// TIA Portal V15.1 export
// export: Created 2024-06-21T08:40:52.8738255Z, ExportSetting WithDefaults, DisplayName Totally Integrated Automation Portal, DisplayVersion V15.1 Update 5, DisplayName TIA Portal Openness, DisplayVersion V15.1 Update 5, DisplayName SINAMICS Startdrive Advanced, DisplayVersion V15.1, DisplayName G130, G150, S120, S150, SINAMICS MV, S210, DisplayVersion V15.1, DisplayName G110M, G120, G120C, G120D, G120P, DisplayVersion V15.1, DisplayName STEP 7 Professional, DisplayVersion V15.1 Update 5, DisplayName STEP 7 Safety, DisplayVersion V15.1, DisplayName WinCC Professional, DisplayVersion V15.1 Update 5, DisplayName SIMATIC Visualization Architect, DisplayVersion V15.1
FUNCTION_BLOCK "LGeneralReverse"   // FB1103, FBD
TITLE = LGeneralReverse
{ S7_Optimized_Access := 'TRUE' }
VERSION : 0.1
// stored: AutoNumber false, IsIECCheckEnabled false, IsRetainMemResEnabled false, MemoryReserve 100, SetENOAutomatically False, UDAEnableTagReadback false
   VAR_INPUT
      I_GeneralReverseSw { ExternalAccessible := 'False'; ExternalVisible := 'False'; ExternalWritable := 'False'} : Bool;   // General reverse switch
      I_FbkContactorFwd { ExternalAccessible := 'False'; ExternalVisible := 'False'; ExternalWritable := 'False'} : Bool;   // Feedback contactor Forward
      I_FbkContactorBwd { ExternalAccessible := 'False'; ExternalVisible := 'False'; ExternalWritable := 'False'} : Bool;   // Feedback contactor Backward
      I_EnableAlarm { ExternalAccessible := 'False'; ExternalVisible := 'False'; ExternalWritable := 'False'} : Bool;   // Enable alarm / Enable Alarm
      I_ResetFbkAlarm { ExternalAccessible := 'False'; ExternalVisible := 'False'; ExternalWritable := 'False'} : Bool;   // Reset feedback alarm / Alarm reset pushbutton is activated
      C_FeedbackUsed { ExternalAccessible := 'False'; ExternalVisible := 'False'; ExternalWritable := 'False'} : Bool;   // Config Feedback used
   END_VAR
   VAR_OUTPUT
      O_ContactorFwd { ExternalAccessible := 'False'; ExternalVisible := 'False'; ExternalWritable := 'False'} : Bool;   // Activate low speed contactor / Activate Forward contactor
      O_ContactorBwd { ExternalAccessible := 'False'; ExternalVisible := 'False'; ExternalWritable := 'False'} : Bool;   // Activate High Speed contactor / Activate Backward contactor
      O_GenRevSw { ExternalAccessible := 'False'; ExternalVisible := 'False'; ExternalWritable := 'False'} : Bool;   // General reverse switch
      O_AlarmABCondition { ExternalAccessible := 'False'; ExternalVisible := 'False'; ExternalWritable := 'False'} : Bool;   // Alarm AB Condition
      O_AlarmA { ExternalAccessible := 'False'; ExternalVisible := 'False'; ExternalWritable := 'False'} : Bool;   // Alarm A
      O_AlarmB { ExternalAccessible := 'False'; ExternalVisible := 'False'; ExternalWritable := 'False'} : Bool;   // Alarm B
      O_AlarmC { ExternalAccessible := 'False'; ExternalVisible := 'False'; ExternalWritable := 'False'} : Bool;   // Alarm C
      O_AlarmD { ExternalAccessible := 'False'; ExternalVisible := 'False'; ExternalWritable := 'False'} : Bool;   // Alarm D
      H_AlarmDWord { ExternalAccessible := 'False'; ExternalVisible := 'False'; ExternalWritable := 'False'} : DWord;   // Alarm Word
   END_VAR
   VAR_IN_OUT
      IO_Modes : "Modes";   // Modes
      H_HMI : "H_HMI";   // Icon Animation
      H_GeneralReverse : "H_GeneralReverse";   // Animation
   END_VAR
   VAR
      AB_FbkContactorFwd { ExternalAccessible := 'False'; ExternalVisible := 'False'; ExternalWritable := 'False'} : Bool;   // Feedback error Contactor Forward
      AB_FbkContactorBwd { ExternalAccessible := 'False'; ExternalVisible := 'False'; ExternalWritable := 'False'} : Bool;   // Feedback error Contactor Backward
      AB_GeneralReverseSw { ExternalAccessible := 'False'; ExternalVisible := 'False'; ExternalWritable := 'False'} : Bool;   // General reverse is activated
      AC_GeneralReverseSw { ExternalAccessible := 'False'; ExternalVisible := 'False'; ExternalWritable := 'False'} : Bool;   // General reverse Switch is active
      FbkContactorFwdAlmCond { ExternalAccessible := 'False'; ExternalVisible := 'False'; ExternalWritable := 'False'} : Bool;   // Motor protection alarm condition / Motor protection Alarm condition / Feedback Contactor Forward Alarm condition
      FbkContactorBwdAlmCond { ExternalAccessible := 'False'; ExternalVisible := 'False'; ExternalWritable := 'False'} : Bool;   // Motor protection alarm condition / Motor protection Alarm condition / Feedback Contactor Backward Alarm condition
      AlarmA { ExternalAccessible := 'False'; ExternalVisible := 'False'; ExternalWritable := 'False'} : Bool;   // Alarm A
      AlarmB { ExternalAccessible := 'False'; ExternalVisible := 'False'; ExternalWritable := 'False'} : Bool;   // Alarm B
      AlarmC { ExternalAccessible := 'False'; ExternalVisible := 'False'; ExternalWritable := 'False'} : Bool;   // Alarm C
      AlarmD { ExternalAccessible := 'False'; ExternalVisible := 'False'; ExternalWritable := 'False'} : Bool;   // Alarm D
      AlarmABCondition { ExternalAccessible := 'False'; ExternalVisible := 'False'; ExternalWritable := 'False'} : Bool;   // Alarm AB Condition
      ContactorFwd { ExternalAccessible := 'False'; ExternalVisible := 'False'; ExternalWritable := 'False'} : Bool;   // Activate low speed contactor / Activate Forward contactor
      ContactorBwd { ExternalAccessible := 'False'; ExternalVisible := 'False'; ExternalWritable := 'False'} : Bool;   // Activate High Speed contactor / Activate Backward contactor
      _TimerInit { ExternalAccessible := 'False'; ExternalVisible := 'False'; ExternalWritable := 'False'} : TON_TIME;   // Timer
      _TimerContactorFwd { ExternalAccessible := 'False'; ExternalVisible := 'False'; ExternalWritable := 'False'} : TON_TIME;   // Timer
      _TimerContactorBwd { ExternalAccessible := 'False'; ExternalVisible := 'False'; ExternalWritable := 'False'} : TON_TIME;   // Timer
      _TimerContactorFwdFbk { ExternalAccessible := 'False'; ExternalVisible := 'False'; ExternalWritable := 'False'} : TON_TIME;   // Timer
      _TimerContactorBwdFbk { ExternalAccessible := 'False'; ExternalVisible := 'False'; ExternalWritable := 'False'} : TON_TIME;   // Timer
      _ContactorFwdFbk { ExternalAccessible := 'False'; ExternalVisible := 'False'; ExternalWritable := 'False'} : "L1AlarmMultiIn";   // FB
      _ContactorBwdFbk { ExternalAccessible := 'False'; ExternalVisible := 'False'; ExternalWritable := 'False'} : "L1AlarmMultiIn";   // FB
      Edge { ExternalAccessible := 'False'; ExternalVisible := 'False'; ExternalWritable := 'False'} : Array[1..10] of Bool;   // Edge
   END_VAR
   VAR_TEMP   // added for the SCL form of the ladder/FBD networks
      _w1 : Bool;
      _w2 : Bool;
   END_VAR
BEGIN

REGION Network 1: ****2.1 - Enable Alarms **** Enable Contactor Forward Feedback Alarm
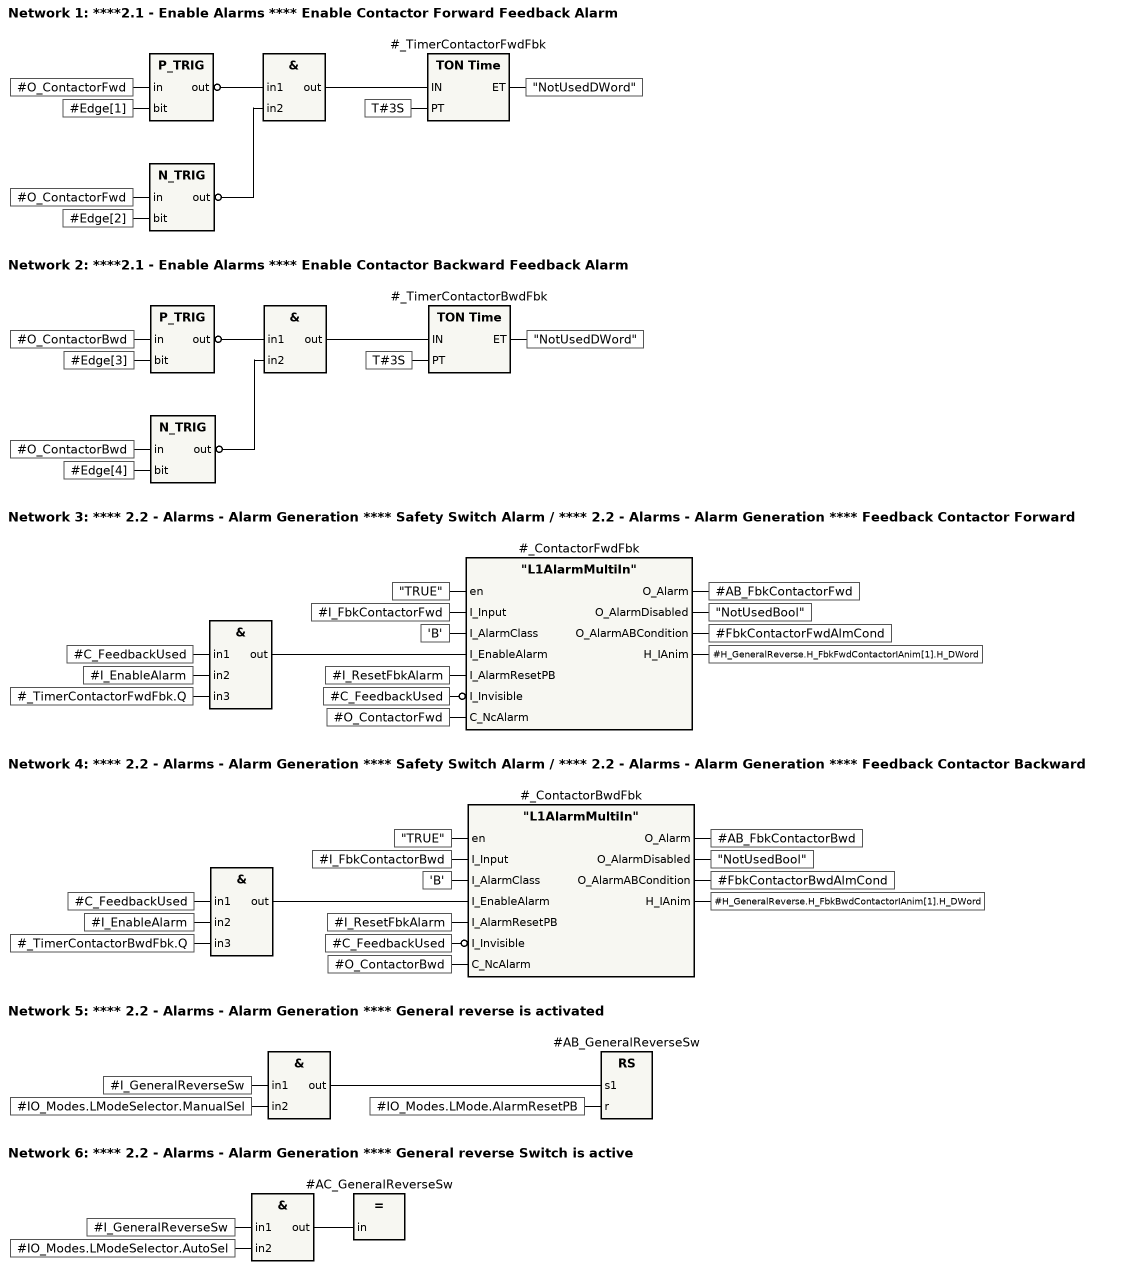
   #_w1 := #O_ContactorFwd AND NOT #Edge[1];   // rising edge
   #Edge[1] := #O_ContactorFwd;
   #_w2 := NOT #O_ContactorFwd AND #Edge[2];   // falling edge
   #Edge[2] := #O_ContactorFwd;
   #_TimerContactorFwdFbk(IN := NOT #_w1 AND NOT #_w2, PT := T#3S, ET => "NotUsedDWord");   // TON
END_REGION

REGION Network 2: ****2.1 - Enable Alarms **** Enable Contactor Backward Feedback Alarm
   #_w1 := #O_ContactorBwd AND NOT #Edge[3];   // rising edge
   #Edge[3] := #O_ContactorBwd;
   #_w2 := NOT #O_ContactorBwd AND #Edge[4];   // falling edge
   #Edge[4] := #O_ContactorBwd;
   #_TimerContactorBwdFbk(IN := NOT #_w1 AND NOT #_w2, PT := T#3S, ET => "NotUsedDWord");   // TON
END_REGION

REGION Network 3: **** 2.2 - Alarms - Alarm Generation **** Safety Switch Alarm / **** 2.2 - Alarms - Alarm Generation **** Feedback Contactor Forward
   // Safety Switch Alarm / Feedback error Contactor Forward
   IF "TRUE" THEN
       #_ContactorFwdFbk(I_Input := #I_FbkContactorFwd,   // "L1AlarmMultiIn"
                         I_AlarmClass := 'B',
                         I_EnableAlarm := #C_FeedbackUsed AND #I_EnableAlarm AND #_TimerContactorFwdFbk.Q,
                         I_AlarmResetPB := #I_ResetFbkAlarm,
                         I_Invisible := NOT #C_FeedbackUsed,
                         C_NcAlarm := #O_ContactorFwd,
                         O_Alarm => #AB_FbkContactorFwd,
                         O_AlarmDisabled => "NotUsedBool",
                         O_AlarmABCondition => #FbkContactorFwdAlmCond,
                         H_IAnim => #H_GeneralReverse.H_FbkFwdContactorIAnim[1].H_DWord);
   END_IF;
END_REGION

REGION Network 4: **** 2.2 - Alarms - Alarm Generation **** Safety Switch Alarm / **** 2.2 - Alarms - Alarm Generation **** Feedback Contactor Backward
   // Safety Switch Alarm / Feedback error Contactor Backward
   IF "TRUE" THEN
       #_ContactorBwdFbk(I_Input := #I_FbkContactorBwd,   // "L1AlarmMultiIn"
                         I_AlarmClass := 'B',
                         I_EnableAlarm := #C_FeedbackUsed AND #I_EnableAlarm AND #_TimerContactorBwdFbk.Q,
                         I_AlarmResetPB := #I_ResetFbkAlarm,
                         I_Invisible := NOT #C_FeedbackUsed,
                         C_NcAlarm := #O_ContactorBwd,
                         O_Alarm => #AB_FbkContactorBwd,
                         O_AlarmDisabled => "NotUsedBool",
                         O_AlarmABCondition => #FbkContactorBwdAlmCond,
                         H_IAnim => #H_GeneralReverse.H_FbkBwdContactorIAnim[1].H_DWord);
   END_IF;
END_REGION

REGION Network 5: **** 2.2 - Alarms - Alarm Generation **** General reverse is activated
   IF #IO_Modes.LMode.AlarmResetPB THEN
       #AB_GeneralReverseSw := FALSE;   // RS flip-flop
   END_IF;
   IF #I_GeneralReverseSw AND #IO_Modes.LModeSelector.ManualSel THEN #AB_GeneralReverseSw := TRUE; END_IF;
END_REGION

REGION Network 6: **** 2.2 - Alarms - Alarm Generation **** General reverse Switch is active
   #AC_GeneralReverseSw := #I_GeneralReverseSw AND #IO_Modes.LModeSelector.AutoSel;
END_REGION

REGION Network 7: **** 4.6 - Machine Status - Indication **** Low Speed Contactor Animation / **** 4.6 - Machine Status - Indication **** Forward Contactor Animation
   // Low speed Contactor Animation
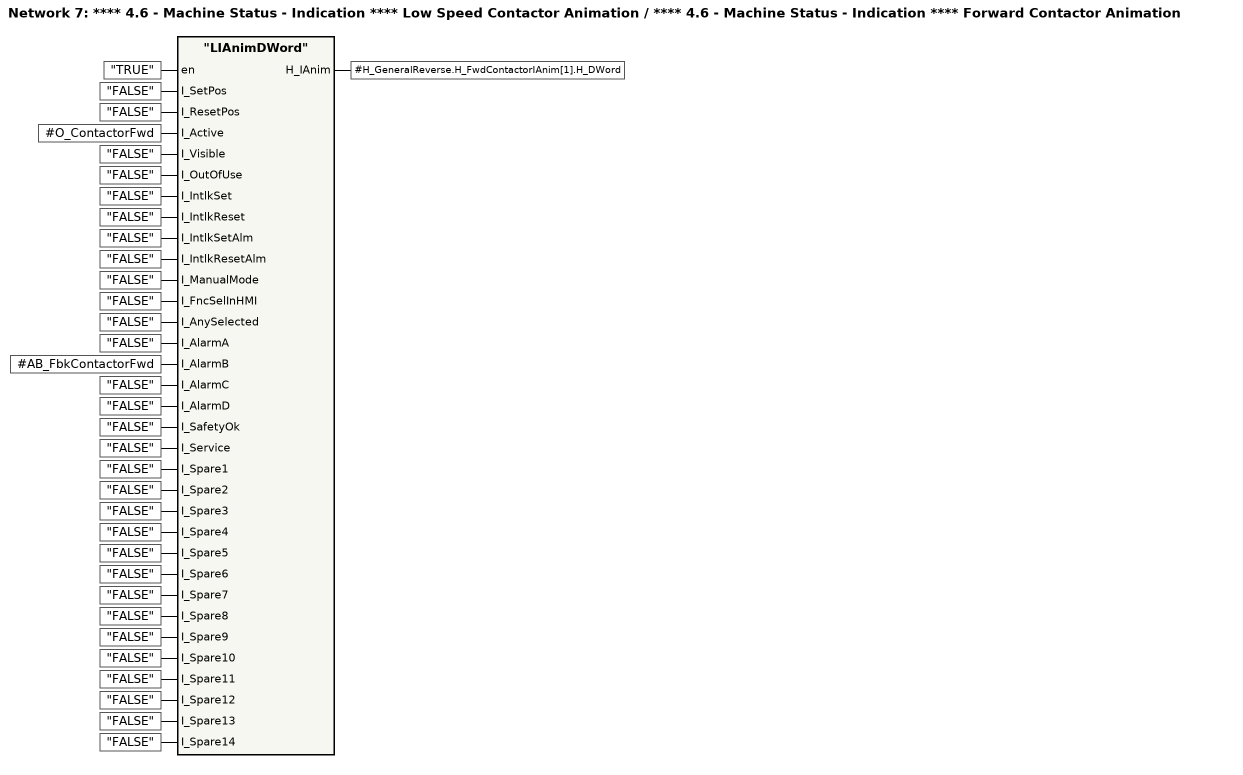
   IF "TRUE" THEN
       "LIAnimDWord"(I_SetPos := "FALSE",
                     I_ResetPos := "FALSE",
                     I_Active := #O_ContactorFwd,
                     I_Visible := "FALSE",
                     I_OutOfUse := "FALSE",
                     I_IntlkSet := "FALSE",
                     I_IntlkReset := "FALSE",
                     I_IntlkSetAlm := "FALSE",
                     I_IntlkResetAlm := "FALSE",
                     I_ManualMode := "FALSE",
                     I_FncSelInHMI := "FALSE",
                     I_AnySelected := "FALSE",
                     I_AlarmA := "FALSE",
                     I_AlarmB := #AB_FbkContactorFwd,
                     I_AlarmC := "FALSE",
                     I_AlarmD := "FALSE",
                     I_SafetyOk := "FALSE",
                     I_Service := "FALSE",
                     I_Spare1 := "FALSE",
                     I_Spare2 := "FALSE",
                     I_Spare3 := "FALSE",
                     I_Spare4 := "FALSE",
                     I_Spare5 := "FALSE",
                     I_Spare6 := "FALSE",
                     I_Spare7 := "FALSE",
                     I_Spare8 := "FALSE",
                     I_Spare9 := "FALSE",
                     I_Spare10 := "FALSE",
                     I_Spare11 := "FALSE",
                     I_Spare12 := "FALSE",
                     I_Spare13 := "FALSE",
                     I_Spare14 := "FALSE",
                     H_IAnim => #H_GeneralReverse.H_FwdContactorIAnim[1].H_DWord);
   END_IF;
END_REGION

REGION Network 8: **** 4.6 - Machine Status - Indication **** High Speed Contactor Animation / **** 4.6 - Machine Status - Indication **** Backward Contactor Animation
   // High Speed Contactor Animation
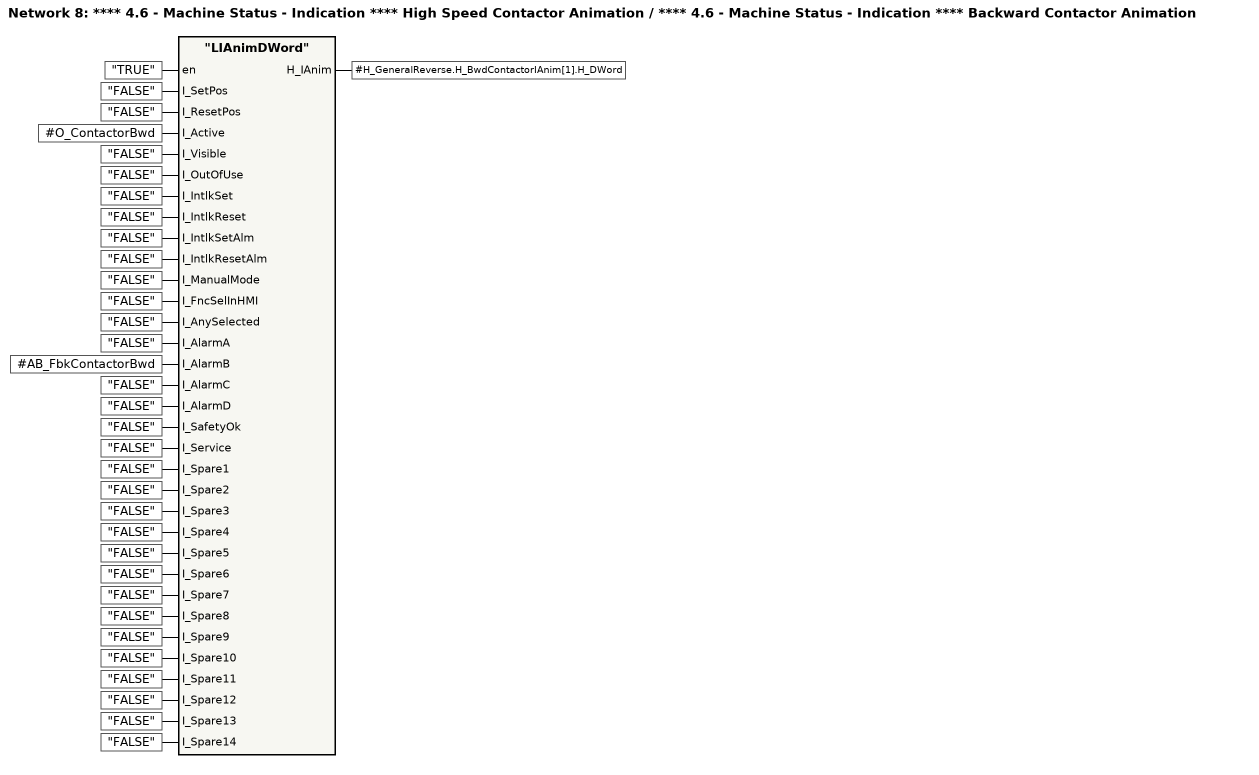
   IF "TRUE" THEN
       "LIAnimDWord"(I_SetPos := "FALSE",
                     I_ResetPos := "FALSE",
                     I_Active := #O_ContactorBwd,
                     I_Visible := "FALSE",
                     I_OutOfUse := "FALSE",
                     I_IntlkSet := "FALSE",
                     I_IntlkReset := "FALSE",
                     I_IntlkSetAlm := "FALSE",
                     I_IntlkResetAlm := "FALSE",
                     I_ManualMode := "FALSE",
                     I_FncSelInHMI := "FALSE",
                     I_AnySelected := "FALSE",
                     I_AlarmA := "FALSE",
                     I_AlarmB := #AB_FbkContactorBwd,
                     I_AlarmC := "FALSE",
                     I_AlarmD := "FALSE",
                     I_SafetyOk := "FALSE",
                     I_Service := "FALSE",
                     I_Spare1 := "FALSE",
                     I_Spare2 := "FALSE",
                     I_Spare3 := "FALSE",
                     I_Spare4 := "FALSE",
                     I_Spare5 := "FALSE",
                     I_Spare6 := "FALSE",
                     I_Spare7 := "FALSE",
                     I_Spare8 := "FALSE",
                     I_Spare9 := "FALSE",
                     I_Spare10 := "FALSE",
                     I_Spare11 := "FALSE",
                     I_Spare12 := "FALSE",
                     I_Spare13 := "FALSE",
                     I_Spare14 := "FALSE",
                     H_IAnim => #H_GeneralReverse.H_BwdContactorIAnim[1].H_DWord);
   END_IF;
END_REGION

REGION Network 9: **** 4.6 - Machine Status - Indication **** Stop Detection Reset / **** 4.6 - Machine Status - Indications **** General Reverse Switch Animation
   // Stop Detection Reset
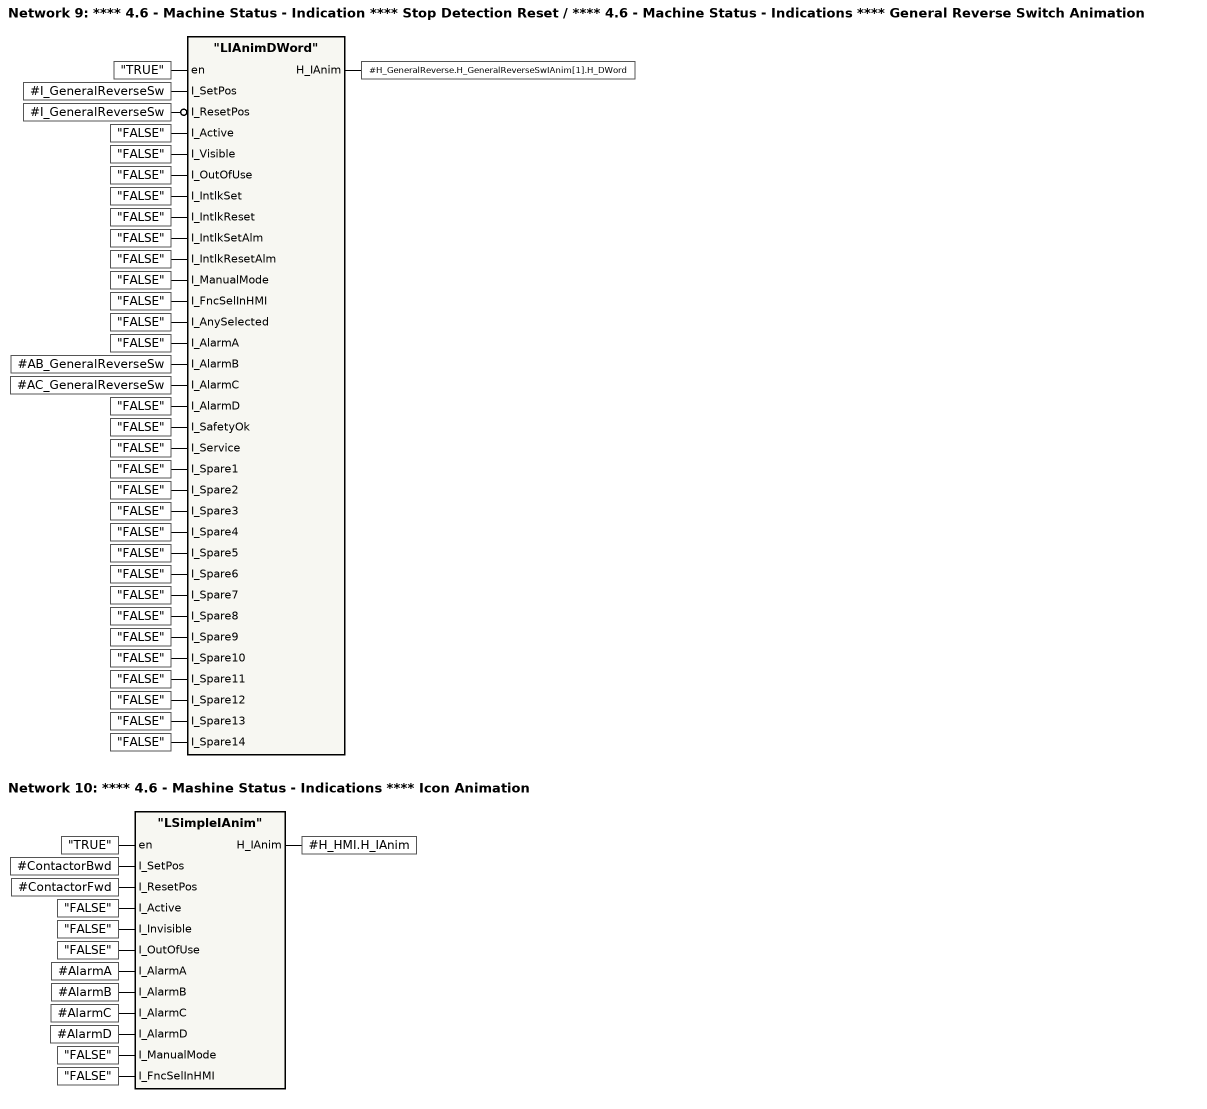
   IF "TRUE" THEN
       "LIAnimDWord"(I_SetPos := #I_GeneralReverseSw,
                     I_ResetPos := NOT #I_GeneralReverseSw,
                     I_Active := "FALSE",
                     I_Visible := "FALSE",
                     I_OutOfUse := "FALSE",
                     I_IntlkSet := "FALSE",
                     I_IntlkReset := "FALSE",
                     I_IntlkSetAlm := "FALSE",
                     I_IntlkResetAlm := "FALSE",
                     I_ManualMode := "FALSE",
                     I_FncSelInHMI := "FALSE",
                     I_AnySelected := "FALSE",
                     I_AlarmA := "FALSE",
                     I_AlarmB := #AB_GeneralReverseSw,
                     I_AlarmC := #AC_GeneralReverseSw,
                     I_AlarmD := "FALSE",
                     I_SafetyOk := "FALSE",
                     I_Service := "FALSE",
                     I_Spare1 := "FALSE",
                     I_Spare2 := "FALSE",
                     I_Spare3 := "FALSE",
                     I_Spare4 := "FALSE",
                     I_Spare5 := "FALSE",
                     I_Spare6 := "FALSE",
                     I_Spare7 := "FALSE",
                     I_Spare8 := "FALSE",
                     I_Spare9 := "FALSE",
                     I_Spare10 := "FALSE",
                     I_Spare11 := "FALSE",
                     I_Spare12 := "FALSE",
                     I_Spare13 := "FALSE",
                     I_Spare14 := "FALSE",
                     H_IAnim => #H_GeneralReverse.H_GeneralReverseSwIAnim[1].H_DWord);
   END_IF;
END_REGION

REGION Network 10: **** 4.6 - Mashine Status - Indications **** Icon Animation
   // Icon Animation
   IF "TRUE" THEN
       "LSimpleIAnim"(I_SetPos := #ContactorBwd,
                      I_ResetPos := #ContactorFwd,
                      I_Active := "FALSE",
                      I_Invisible := "FALSE",
                      I_OutOfUse := "FALSE",
                      I_AlarmA := #AlarmA,
                      I_AlarmB := #AlarmB,
                      I_AlarmC := #AlarmC,
                      I_AlarmD := #AlarmD,
                      I_ManualMode := "FALSE",
                      I_FncSelInHMI := "FALSE",
                      H_IAnim => #H_HMI.H_IAnim);
   END_IF;
END_REGION

REGION Network 11: **** 4.6 - Machine status - Indications **** Animation
   // Animation Word 1
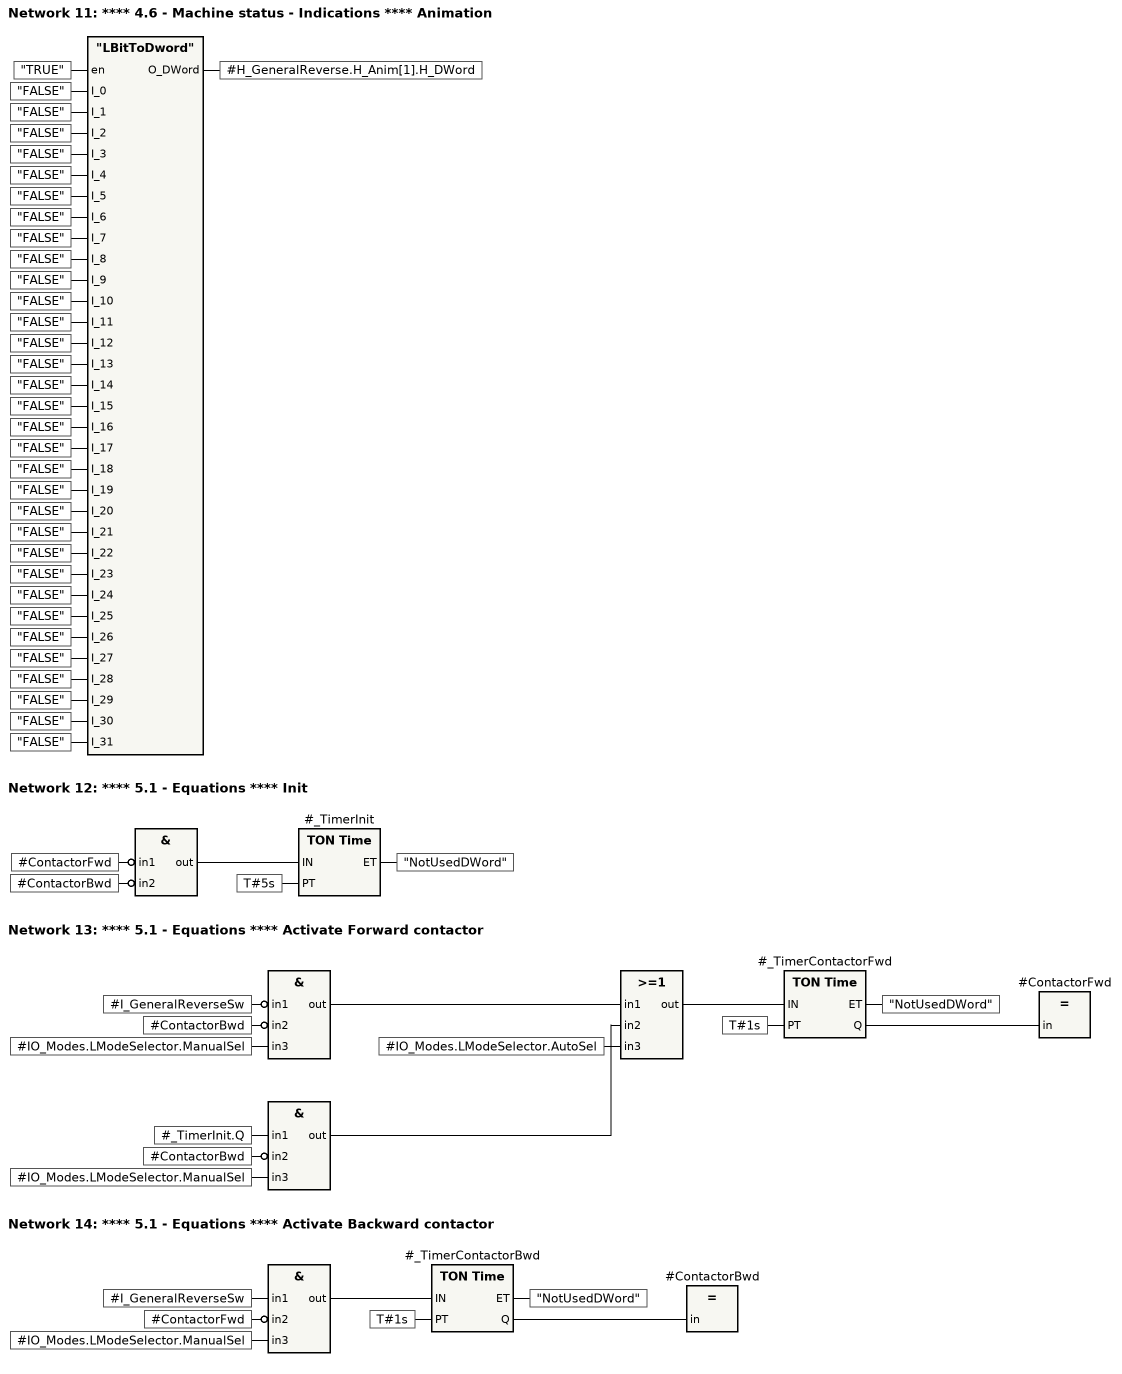
   IF "TRUE" THEN
       "LBitToDword"(I_0 := "FALSE",
                     I_1 := "FALSE",
                     I_2 := "FALSE",
                     I_3 := "FALSE",
                     I_4 := "FALSE",
                     I_5 := "FALSE",
                     I_6 := "FALSE",
                     I_7 := "FALSE",
                     I_8 := "FALSE",
                     I_9 := "FALSE",
                     I_10 := "FALSE",
                     I_11 := "FALSE",
                     I_12 := "FALSE",
                     I_13 := "FALSE",
                     I_14 := "FALSE",
                     I_15 := "FALSE",
                     I_16 := "FALSE",
                     I_17 := "FALSE",
                     I_18 := "FALSE",
                     I_19 := "FALSE",
                     I_20 := "FALSE",
                     I_21 := "FALSE",
                     I_22 := "FALSE",
                     I_23 := "FALSE",
                     I_24 := "FALSE",
                     I_25 := "FALSE",
                     I_26 := "FALSE",
                     I_27 := "FALSE",
                     I_28 := "FALSE",
                     I_29 := "FALSE",
                     I_30 := "FALSE",
                     I_31 := "FALSE",
                     O_DWord => #H_GeneralReverse.H_Anim[1].H_DWord);
   END_IF;
END_REGION

REGION Network 12: **** 5.1 - Equations **** Init
   #_TimerInit(IN := NOT #ContactorFwd AND NOT #ContactorBwd, PT := T#5s, ET => "NotUsedDWord");   // TON
END_REGION

REGION Network 13: **** 5.1 - Equations **** Activate Forward contactor
   #_TimerContactorFwd(IN := (NOT #I_GeneralReverseSw AND NOT #ContactorBwd AND #IO_Modes.LModeSelector.ManualSel) OR (#_TimerInit.Q AND NOT #ContactorBwd AND #IO_Modes.LModeSelector.ManualSel) OR #IO_Modes.LModeSelector.AutoSel,   // TON
                       PT := T#1s,
                       ET => "NotUsedDWord");
   #ContactorFwd := #_TimerContactorFwd.Q;
END_REGION

REGION Network 14: **** 5.1 - Equations **** Activate Backward contactor
   #_TimerContactorBwd(IN := #I_GeneralReverseSw AND NOT #ContactorFwd AND #IO_Modes.LModeSelector.ManualSel,   // TON
                       PT := T#1s,
                       ET => "NotUsedDWord");
   #ContactorBwd := #_TimerContactorBwd.Q;
END_REGION

REGION Network 15: **** 8 - Outputs **** Alarm AB Condition
   // Alarm AB Condition
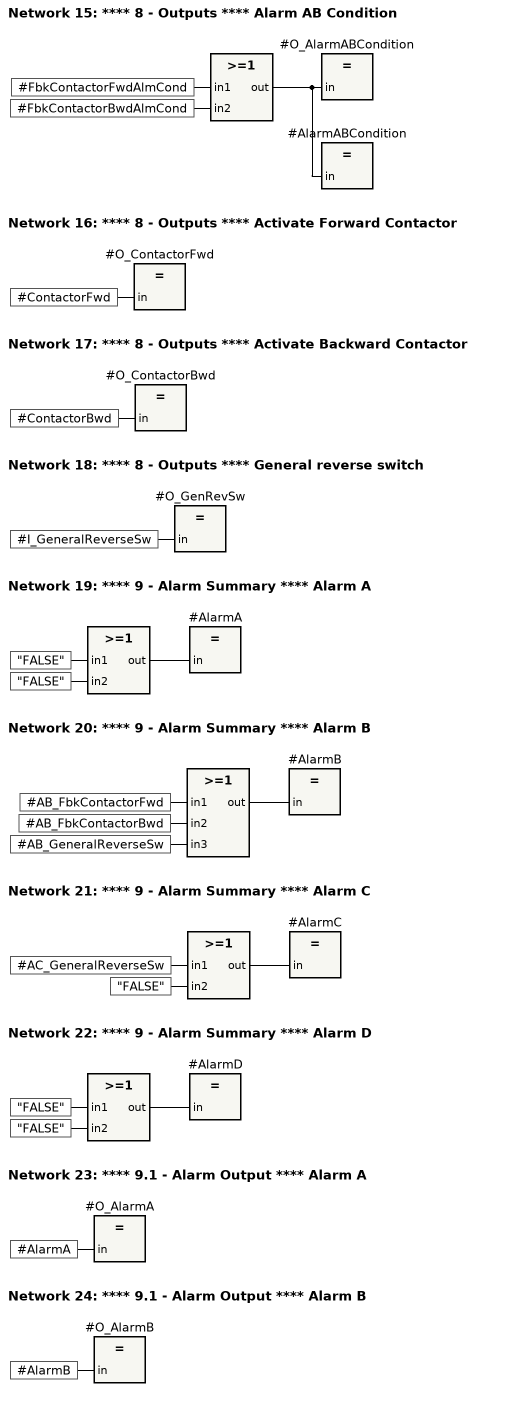
   #O_AlarmABCondition := #FbkContactorFwdAlmCond OR #FbkContactorBwdAlmCond;
   #AlarmABCondition := #O_AlarmABCondition;
END_REGION

REGION Network 16: **** 8 - Outputs **** Activate Forward Contactor
   #O_ContactorFwd := #ContactorFwd;
END_REGION

REGION Network 17: **** 8 - Outputs **** Activate Backward Contactor
   #O_ContactorBwd := #ContactorBwd;
END_REGION

REGION Network 18: **** 8 - Outputs **** General reverse switch
   #O_GenRevSw := #I_GeneralReverseSw;
END_REGION

REGION Network 19: **** 9 - Alarm Summary **** Alarm A
   // Alarm A
   #AlarmA := "FALSE" OR "FALSE";
END_REGION

REGION Network 20: **** 9 - Alarm Summary **** Alarm B
   // Alarm B
   #AlarmB := #AB_FbkContactorFwd OR #AB_FbkContactorBwd OR #AB_GeneralReverseSw;
END_REGION

REGION Network 21: **** 9 - Alarm Summary **** Alarm C
   // Alarm C
   #AlarmC := #AC_GeneralReverseSw OR "FALSE";
END_REGION

REGION Network 22: **** 9 - Alarm Summary **** Alarm D
   // Alarm D
   #AlarmD := "FALSE" OR "FALSE";
END_REGION

REGION Network 23: **** 9.1 - Alarm Output **** Alarm A
   // Alarm A
   #O_AlarmA := #AlarmA;
END_REGION

REGION Network 24: **** 9.1 - Alarm Output **** Alarm B
   // Alarm B
   #O_AlarmB := #AlarmB;
END_REGION

REGION Network 25: **** 9.1 - Alarm Output **** Alarm C
   // Alarm C
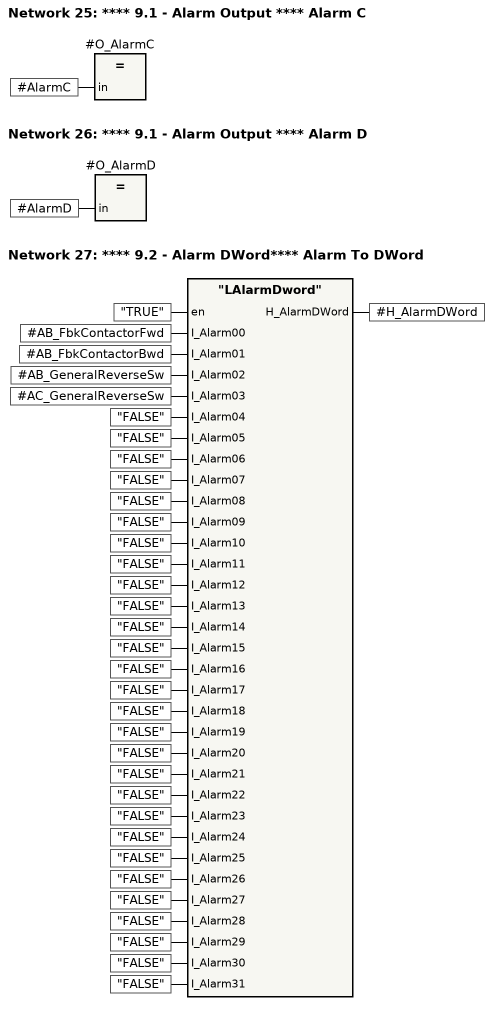
   #O_AlarmC := #AlarmC;
END_REGION

REGION Network 26: **** 9.1 - Alarm Output **** Alarm D
   // Alarm D
   #O_AlarmD := #AlarmD;
END_REGION

REGION Network 27: **** 9.2 - Alarm DWord**** Alarm To DWord
   // Alarm To DWord
   IF "TRUE" THEN
       "LAlarmDword"(I_Alarm00 := #AB_FbkContactorFwd,
                     I_Alarm01 := #AB_FbkContactorBwd,
                     I_Alarm02 := #AB_GeneralReverseSw,
                     I_Alarm03 := #AC_GeneralReverseSw,
                     I_Alarm04 := "FALSE",
                     I_Alarm05 := "FALSE",
                     I_Alarm06 := "FALSE",
                     I_Alarm07 := "FALSE",
                     I_Alarm08 := "FALSE",
                     I_Alarm09 := "FALSE",
                     I_Alarm10 := "FALSE",
                     I_Alarm11 := "FALSE",
                     I_Alarm12 := "FALSE",
                     I_Alarm13 := "FALSE",
                     I_Alarm14 := "FALSE",
                     I_Alarm15 := "FALSE",
                     I_Alarm16 := "FALSE",
                     I_Alarm17 := "FALSE",
                     I_Alarm18 := "FALSE",
                     I_Alarm19 := "FALSE",
                     I_Alarm20 := "FALSE",
                     I_Alarm21 := "FALSE",
                     I_Alarm22 := "FALSE",
                     I_Alarm23 := "FALSE",
                     I_Alarm24 := "FALSE",
                     I_Alarm25 := "FALSE",
                     I_Alarm26 := "FALSE",
                     I_Alarm27 := "FALSE",
                     I_Alarm28 := "FALSE",
                     I_Alarm29 := "FALSE",
                     I_Alarm30 := "FALSE",
                     I_Alarm31 := "FALSE",
                     H_AlarmDWord => #H_AlarmDWord);
   END_IF;
END_REGION
END_FUNCTION_BLOCK
